{attribute 'linkalways'} 
{attribute 'no_explicit_call' := 'This FB is a CLASS and must be accessed using methods or properties'}
{attribute 'enable_dynamic_creation'}
FUNCTION_BLOCK _LWORD EXTENDS NumericDatatypeBase
VAR
	localData : LWORD;
	activeData : REFERENCE TO LWORD REF= localData;
END_VAR

PROPERTY PUBLIC Address : PVOID
GET
Address := ADR(activeData);
END_GET
END_PROPERTY

METHOD PUBLIC ClearReference
VAR_INPUT
END_VAR
activeData REF= localData;
END_METHOD

METHOD PUBLIC Clone : I_Datatype
VAR
    pClone : POINTER TO _LWORD;
END_VAR
pClone := __NEW(_LWORD(InitialValue := Value));
Clone := pClone^;
END_METHOD

METHOD FB_init : BOOL
VAR_INPUT
	bInitRetains : BOOL; // if TRUE, the retain variables are initialized (warm start / cold start)
	bInCopyCode : BOOL;  // if TRUE, the instance afterwards gets moved WORDo the copy code (online change)
	InitialValue : LWORD;
END_VAR
localData := InitialValue;
END_METHOD

PROPERTY PUBLIC IsEven : BOOL
GET
IsEven := (Value mod 2) = 0;
END_GET
END_PROPERTY

PROPERTY PUBLIC IsFloat : BOOL
GET
IsFloat := FALSE;
END_GET
END_PROPERTY

PROPERTY PUBLIC IsSigned : BOOL
GET
IsSigned := FALSE;
END_GET
END_PROPERTY

METHOD PUBLIC MakeReferenceTo
VAR_INPUT
	ReferenceTarget : REFERENCE TO LWORD;
END_VAR
activeData REF= ReferenceTarget;
END_METHOD

PROPERTY PUBLIC MaxValue : LWORD
GET
MaxValue :=  DatatypeLimits.LWORD_MAX_VALUE;
END_GET
END_PROPERTY

PROPERTY PUBLIC MinValue : LWORD
GET
MinValue := DatatypeLimits.LWORD_MIN_VALUE;
END_GET
END_PROPERTY

METHOD PROTECTED SerializeMaxValue
VAR_INPUT
	Serializer : I_Serializer;
END_VAR
Serializer.AddLword(MaxValue);
END_METHOD

METHOD PROTECTED SerializeMinValue
VAR_INPUT
	Serializer : I_Serializer;
END_VAR
Serializer.AddLword(MinValue);
END_METHOD

METHOD PUBLIC SerializeWith
VAR_INPUT
	Serializer : I_Serializer;
END_VAR
Serializer.AddLword(activeData);
END_METHOD

PROPERTY PUBLIC Size : UDINT
GET
Size := SIZEOF(activeData);
END_GET
END_PROPERTY

METHOD TryDeserializeFrom : BOOL
VAR_INPUT
	Deserializer : I_Deserializer;
	Feedback : I_DeserializerFeedback;
END_VAR
TryDeserializeFrom := Deserializer.TryGetLword(activeData, Feedback);
END_METHOD

METHOD TryMakeReferenceTo : BOOL
VAR_INPUT
	Target : I_Datatype;
END_VAR
VAR
	pTargetData : POINTER TO LWORD;
END_VAR
IF NOT (Target.TypeName = TypeName) THEN
	RETURN;
END_IF

pTargetData := Target.Address;
activeData REF= pTargetData^;
TryMakeReferenceTo := TRUE;
END_METHOD

PROPERTY PUBLIC TypeName : T_MAXSTRING
GET
TypeName := 'LWORD';
END_GET
END_PROPERTY

PROPERTY PUBLIC Value : REFERENCE TO LWORD
GET
Value REF= activeData;
END_GET
END_PROPERTY

END_FUNCTION_BLOCK

(* stored: Version 1.1.0.1, ProductVersion 3.1.4024.13
   POU _LWORD: Id {222c1fd0-7220-4b1a-89da-6ed583eaaa15}, SpecialFunc None
   Folder Constructor: Id {131450bd-6664-43d6-a9ed-cdfb6bd3565b}
   Folder Protected: Id {59e42608-a20c-4e49-b9ed-d0540691eef7}
   Property Address: Id {81e4bc0f-3f27-4971-a04b-33a72acbc3e4}
   Get Get: Id {10583fe8-8424-4749-9ca3-e2913d2cc275}
   Method ClearReference: Id {7623f491-f071-4d4a-8fb1-18dff4157132}
   Method Clone: Id {db8b75a8-d11e-476c-b5c9-f47df3d8e7a2}
   Method FB_init: Id {0af42890-492b-4f8f-a6e1-0dcc21c668f2}
   Property IsEven: Id {10486f73-2e55-0816-04cd-31baed6be3fc}
   Get Get: Id {11c1b12a-f4eb-00da-1820-2207ed7e53c6}
   Property IsFloat: Id {6c21dc09-f552-4e54-a942-18a3b753fea0}
   Get Get: Id {d0858414-1304-4cca-8f9d-feb5e8414ac4}
   Property IsSigned: Id {2d2483d8-6836-4bf2-bdf7-90f8a9ca9a41}
   Get Get: Id {fe02f237-9497-40cd-9764-69e53fe63bc2}
   Method MakeReferenceTo: Id {50b83421-15b3-4123-b64a-cfd32145299e}
   Property MaxValue: Id {04df833c-ad46-484d-994f-83a287b8f654}
   Get Get: Id {59340785-85d0-43a7-9d3e-737c333d6255}
   Property MinValue: Id {cc907cc4-91d6-4b69-9d2d-8c3d10842232}
   Get Get: Id {be29745a-c42d-48c3-bbd7-6dea2b883184}
   Method SerializeMaxValue: Id {aca5f6f7-3cbf-4c1c-9896-504b1b3e1b9c}
   Method SerializeMinValue: Id {d3b94d44-d648-45e0-9ffa-3a6770072a97}
   Method SerializeWith: Id {e06bb6cf-2463-4639-a39a-1159511afe2f}
   Property Size: Id {e31c3e68-0f85-4a76-b0a6-44e2826fd0db}
   Get Get: Id {719ece08-08cc-4e40-8d45-1c56d99bc000}
   Method TryDeserializeFrom: Id {b754c233-9c98-4943-83e3-68e869679f5e}
   Method TryMakeReferenceTo: Id {8809cb77-5ffe-4f66-9f35-55da27978f6e}
   Property TypeName: Id {0b5d2a3c-4d2e-4f82-85c0-9844136e0df8}
   Get Get: Id {127c7ccb-358c-49db-b9ae-0e2c2c50519b}
   Property Value: Id {bfff94ba-74bc-4235-8193-f4c8306c3a0c}
   Get Get: Id {a9628c75-9e11-4d99-9a0e-452850106776} *)
